TYPE EL6001_COM_Inputs :
STRUCT
	{attribute addProperty Name "Status"}
	Status AT %I* : EL6001_Status;
	{attribute addProperty Name "Data"}
	Data  AT %I* : ARRAY[0..21] OF USINT;
END_STRUCT
END_TYPE

(* stored: Version 1.1.0.1, ProductVersion 3.1.4024.9
   DUT EL6001_COM_Inputs: Id {fe169e60-688b-0262-363a-75d27eee1824} *)
